(* Logix 5000 project; controller ecust2024 vendor 1 type 14 code 108 rev 30.11; software revision 30.00 *)

TASK MainTask (continuous, watchdog 500 ms) : MainProgram, My_Equipment_Phase

MODULES
   Local : vendor 1 type 14 code 108 (Compact 0, rev 30.11)
      K5500 : 2198-H008-ERS (Ethernet 192.168.1.31, rev 7.13, MotionSync RPI 1 ms, MotionDiagnostics RPI 1 ms)
END_MODULES

ADD_ON_INSTRUCTION AOI   (* revision 1.0 *)
VAR_INPUT
   Start : BOOL; {access None, required}
   Stop : BOOL; {required}
END_VAR
VAR_OUTPUT
   LampOut : BOOL; {access Read Only, required}
END_VAR
VAR_INPUT
   Timer1Set : DINT; {required}
   Timer2Set : DINT; {required}
   Timer3Set : DINT; {required}
   TotalTimerSet : DINT; {required}
END_VAR
VAR
   SysGo : BOOL; {access None}
   Timer_1 : TIMER; {access None}
   Timer_2 : TIMER; {access None}
   Timer_3 : TIMER; {access None}
   Timer_T : TIMER; {access None}
END_VAR

ROUTINE Logic   (* ladder *)
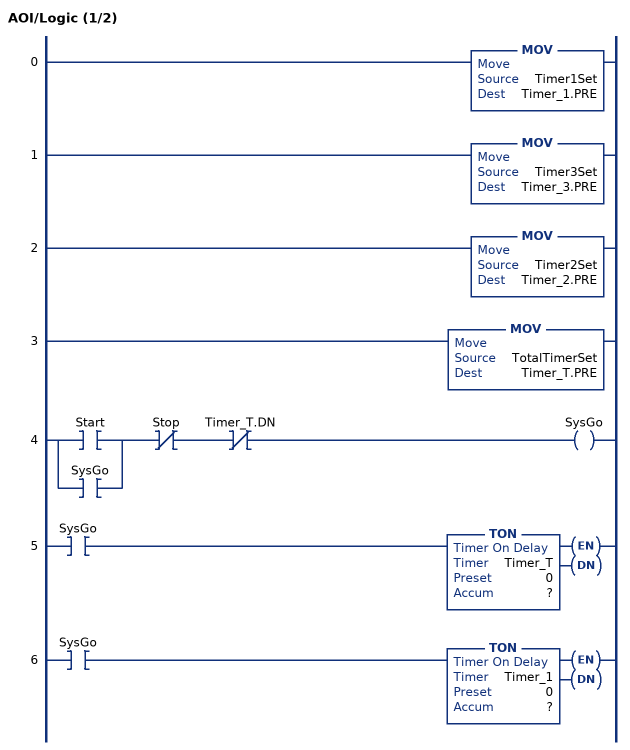
   0: MOV(Timer1Set,Timer_1.PRE);
   1: MOV(Timer3Set,Timer_3.PRE);
   2: MOV(Timer2Set,Timer_2.PRE);
   3: MOV(TotalTimerSet,Timer_T.PRE);
   4: [XIC(Start) ,XIC(SysGo) ]XIO(Stop)XIO(Timer_T.DN)OTE(SysGo);
   5: XIC(SysGo)TON(Timer_T,?,?);
   6: XIC(SysGo)TON(Timer_1,?,?);
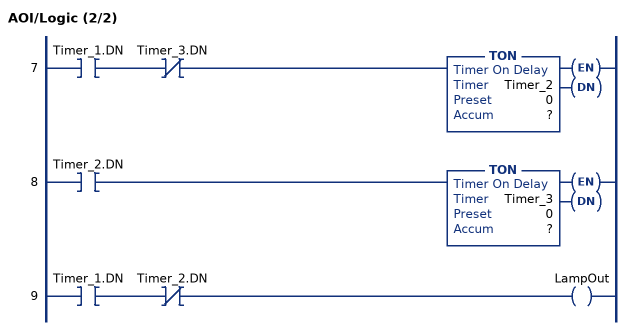
   7: XIC(Timer_1.DN)XIO(Timer_3.DN)TON(Timer_2,?,?);
   8: XIC(Timer_2.DN)TON(Timer_3,?,?);
   9: XIC(Timer_1.DN)XIO(Timer_2.DN)OTE(LampOut);
END_ROUTINE
END_ADD_ON_INSTRUCTION

ADD_ON_INSTRUCTION LED_control   (* revision 1.0 *)
VAR_INPUT
   span : DINT; {required}
END_VAR
VAR_OUTPUT
   LED_start : BOOL; {access Read Only, visible}
END_VAR
VAR_INPUT
   Stop : BOOL; {required}
END_VAR
VAR
   delay1 : TIMER; {access None}
   delay2 : TIMER; {access None}
END_VAR

ROUTINE Logic   (* ladder *)
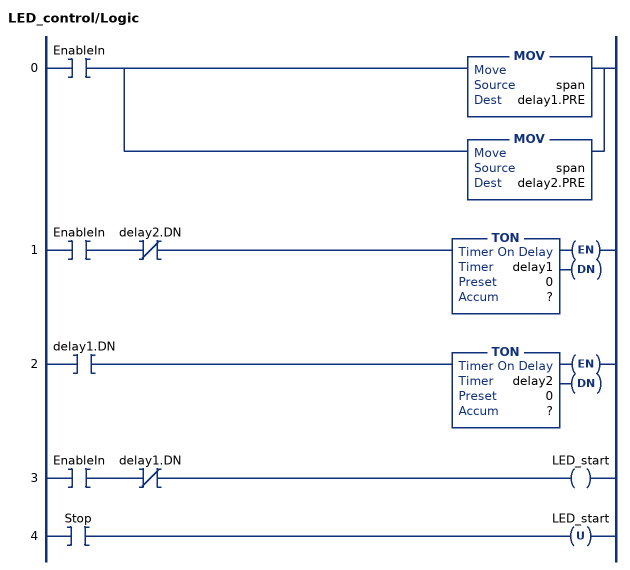
   0: XIC(EnableIn)[MOV(span,delay1.PRE) ,MOV(span,delay2.PRE) ];
   1: XIC(EnableIn)XIO(delay2.DN)TON(delay1,?,?);
   2: XIC(delay1.DN)TON(delay2,?,?);
   3: XIC(EnableIn)XIO(delay1.DN)OTE(LED_start);
   4: XIC(Stop)OTU(LED_start);
END_ROUTINE
END_ADD_ON_INSTRUCTION

ADD_ON_INSTRUCTION OneKey   (* revision 1.0 *)
VAR_INPUT
   Button : BOOL; {required}
END_VAR
VAR_OUTPUT
   On : BOOL; {visible}
   Off : BOOL; {visible}
END_VAR
VAR_INPUT
   Pos1 : DINT; {required}
   Pos2 : DINT; {required}
   speed : DINT; {required}
   Stop_Time : DINT; {required}
END_VAR
VAR_OUTPUT
   Stop1 : BOOL; {access Read Only, visible}
   clockwise : BOOL; {access Read Only, visible}
   anticlockwise : BOOL; {access Read Only, visible}
   Stop2 : BOOL; {access Read Only, visible}
END_VAR
VAR
   delay1 : TIMER; {access None}
   delay2 : TIMER; {access None}
   delay3 : TIMER; {access None}
   oneshot1 : DINT; {access None}
   stop_1 : BOOL; {access None}
   stop_2 : BOOL; {access None}
   Start_state : BOOL; {access None}
   delay4 : TIMER := (PRE := 500); {access None}
END_VAR

ROUTINE Logic   (* ladder *)
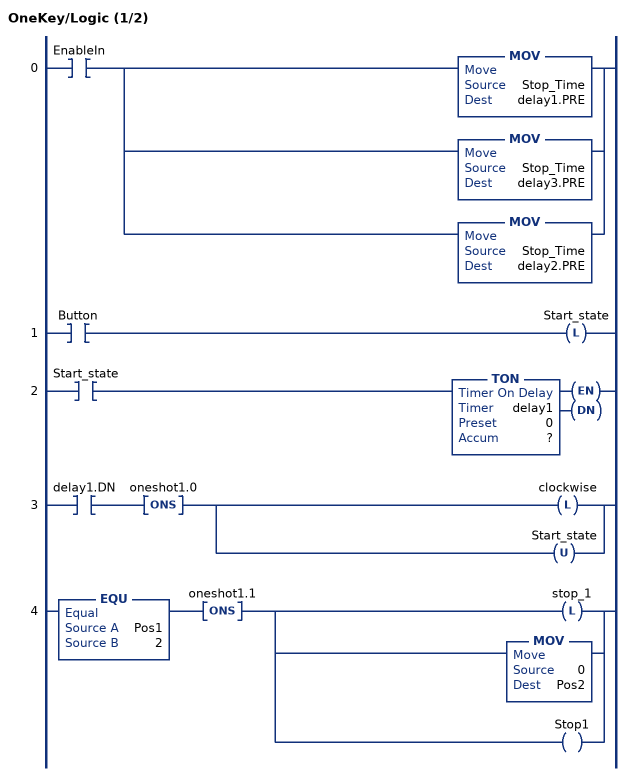
   0: XIC(EnableIn)[MOV(Stop_Time,delay1.PRE) ,MOV(Stop_Time,delay3.PRE) ,MOV(Stop_Time,delay2.PRE) ];
   1: XIC(Button)OTL(Start_state);
   2: XIC(Start_state)TON(delay1,?,?);
   3: XIC(delay1.DN)ONS(oneshot1.0)[OTL(clockwise) ,OTU(Start_state) ];
   4: EQU(Pos1,2)ONS(oneshot1.1)[OTL(stop_1) ,MOV(0,Pos2) ,OTE(Stop1) ];
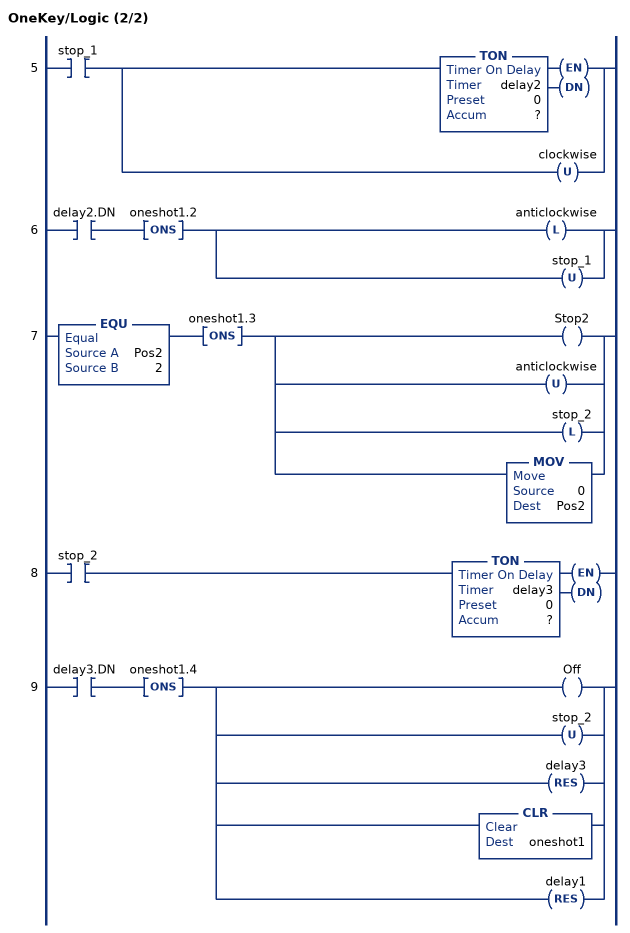
   5: XIC(stop_1)[TON(delay2,?,?) ,OTU(clockwise) ];
   6: XIC(delay2.DN)ONS(oneshot1.2)[OTL(anticlockwise) ,OTU(stop_1) ];
   7: EQU(Pos2,2)ONS(oneshot1.3)[OTE(Stop2) ,OTU(anticlockwise) ,OTL(stop_2) ,MOV(0,Pos2) ];
   8: XIC(stop_2)TON(delay3,?,?);
   9: XIC(delay3.DN)ONS(oneshot1.4)[OTE(Off) ,OTU(stop_2) ,RES(delay3) ,CLR(oneshot1) ,RES(delay1) ];
END_ROUTINE
END_ADD_ON_INSTRUCTION

VAR_GLOBAL   (* controller tags *)
   A : OneKey;
   ActualVelocity_CMX : REAL;
   alrm : BOOL;
   anticlockwise : MOTION_INSTRUCTION := (FLAGS := 570425344, DN := 1);
   anticlockwise2 : MOTION_INSTRUCTION := (FLAGS := 33554432);
   anticlockwise3 : MOTION_INSTRUCTION;
   anticlockwise_order : BOOL;
   Axis_1 : AXIS_CIP_DRIVE;
   back_spot : BOOL;
   backHole : BOOL;
   backHole1_cmd : BOOL;
   backHole1_cmd1 : BOOL := 1;
   backspot : BOOL;
   BletRound : DINT;
   Change_Hole : BOOL;
   Change_speed : BOOL;
   changespeed : MOTION_INSTRUCTION := (FLAGS := 33554432);
   changespeed1 : MOTION_INSTRUCTION := (FLAGS := 33554432);
   changesppedbutton : BOOL;
   circle_num : INT;
   clockwise1 : MOTION_INSTRUCTION := (FLAGS := 570425344, DN := 1);
   clockwise_order : BOOL;
   Cmd_PowerOff : BOOL;
   Cmd_PowerON : BOOL;
   count1 : COUNTER := (PRE := 3);
   count2 : COUNTER := (PRE := 2);
   count3 : COUNTER := (PRE := 2);
   count4 : COUNTER := (PRE := 2);
   count5 : COUNTER := (PRE := 4);
   count6 : COUNTER := (PRE := 4);
   count7 : COUNTER := (PRE := 2);
   count8 : COUNTER := (PRE := 2, ACC := 1);
   countturns1 : TIMER;
   Direction_Change1 : BOOL;
   Direction_Change2 : BOOL;
   Direction_Change3 : BOOL;
   Direction_Change4 : BOOL;
   Direction_change_state1 : BOOL;
   Direction_change_state2 : BOOL;
   Direction_change_state3 : BOOL;
   dong1 : DINT;
   dong2 : DINT;
   Find_sensor1 : BOOL;
   Find_sensor2 : BOOL;
   Find_sensor3 : BOOL;
   Fwd1_Cmd_CMX : BOOL;
   Holding_Cmd : BOOL;
   Light1 : BOOL;
   Light2 : BOOL;
   Light3 : BOOL;
   LT1 : BOOL;
   LT2 : BOOL;
   LT3 : BOOL;
   MSG_1 : MESSAGE;
        MessageParameters(ServiceCode := 16#004c, LocalElement := Temp_CMX, ...)
   MSG_2 : MESSAGE;
        MessageParameters(ServiceCode := 16#004c, LocalElement := Sensor1, ...)
   MSG_3 : MESSAGE;
        MessageParameters(ServiceCode := 16#004c, LocalElement := Sensor2, ...)
   MSG_4 : MESSAGE;
        MessageParameters(ServiceCode := 16#004c, LocalElement := Sensor3, ...)
   My_Equipment_Phase : PHASE := (State := 64, Idle := 1);
   oneshot : DINT;
   Reset_Cmd : BOOL;
   Restart_Cmd : BOOL;
   result1 : DINT;
   result2 : DINT;
   Rev1_Cmd_CMX : BOOL;
   S : DINT;
   screen_speed : DINT := 1;
   Sensor1 : DINT := 1;
   Sensor1_cmd : BOOL := 1;
   Sensor2 : DINT;
   Sensor2_cmd : BOOL;
   Sensor3 : DINT;
   Sensor3_cmd : BOOL;
   Sensor_cmd : BOOL := 1;
   servo_off : MOTION_INSTRUCTION := (FLAGS := 570425344, DN := 1, STATUS := 2, STATE := 1);
   servo_on : MOTION_INSTRUCTION := (FLAGS := 570425344, DN := 1, STATE := 1);
   setspeed : DINT := 1;
   Start_Cmd : BOOL;
   Start_PB : BOOL;
   StartA : BOOL;
   state_fwd : BOOL;
   state_off : BOOL := 1;
   state_on : BOOL;
   state_rev : BOOL;
   state_stop : BOOL;
   Stop : MOTION_INSTRUCTION := (FLAGS := 704643072, DN := 1, PC := 1);
   Stop1 : MOTION_INSTRUCTION := (FLAGS := 33554432);
   Stop1_Cmd_CMX : BOOL;
   Stop2 : MOTION_INSTRUCTION;
   Stop_Cmd : BOOL;
   Stop_PB : BOOL;
   Temp_CMX : REAL;
   temp_speed : REAL;
   temperature_speed : REAL;
   time1 : TIMER := (PRE := 3000);
   time2 : TIMER := (PRE := 3000);
   time3 : TIMER := (PRE := 3000);
   time4 : TIMER := (PRE := 3000);
   ts : BOOL;
   UM_Motion : MOTION_GROUP;
   wendu_alrm : BOOL;
   xiansudu : REAL;
   yanshi1 : TIMER := (PRE := 500);
   yanshi101 : TIMER := (PRE := 3000);
END_VAR

PROGRAM MainProgram   (* main routine MainRoutine *)
VAR
   circle_count : DINT;
   circle_num1 : DINT;
   count10 : COUNTER := (PRE := 3);
   count11 : COUNTER := (PRE := 3);
   delay1 : TIMER := (PRE := 500);
   delay2 : TIMER := (PRE := 1000);
   delay3 : TIMER := (PRE := 1000);
   delay4 : TIMER := (PRE := 1000);
   LED1 : LED_control;
   LED2 : LED_control;
   LED3 : LED_control;
   LT1_AOI : AOI := (Timer2Set := 2000, Timer3Set := 2000, TotalTimerSet := 30000);
   LT2_AOI : AOI := (Timer1Set := 10000, Timer2Set := 1000, Timer3Set := 1000, TotalTimerSet := 30000);
   LT3_AOI : AOI := (Timer1Set := 20000, Timer2Set := 500, Timer3Set := 500, TotalTimerSet := 30000);
   speed_dec : BOOL;
   speed_inc : BOOL;
   velocity : DINT;
   wait1 : TIMER := (PRE := 10000);
   wait2 : TIMER := (PRE := 10000);
   wait3 : TIMER := (PRE := 10000);
END_VAR

ROUTINE MainRoutine   (* ladder *)
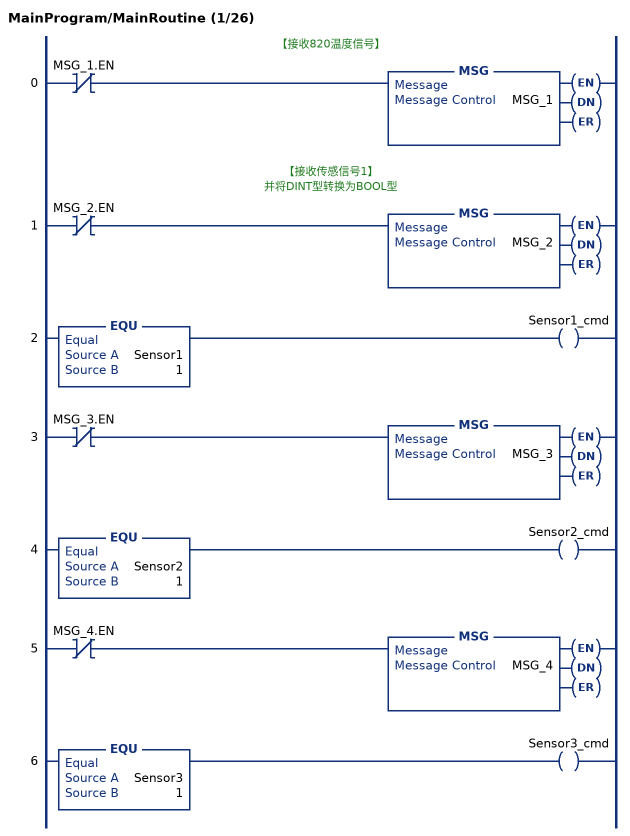
   // 【接收820温度信号】
   0: XIO(MSG_1.EN)MSG(MSG_1);
   // 【接收传感信号1】
   // 并将DINT型转换为BOOL型
   1: XIO(MSG_2.EN)MSG(MSG_2);
   2: EQU(Sensor1,1)OTE(Sensor1_cmd);
   3: XIO(MSG_3.EN)MSG(MSG_3);
   4: EQU(Sensor2,1)OTE(Sensor2_cmd);
   5: XIO(MSG_4.EN)MSG(MSG_4);
   6: EQU(Sensor3,1)OTE(Sensor3_cmd);
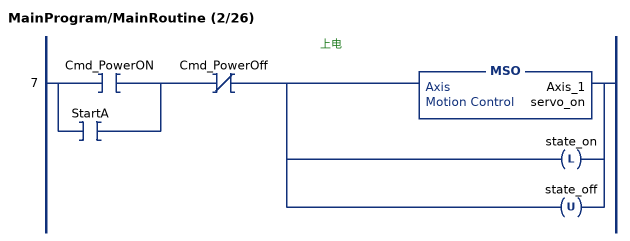
   // 上电
   7: [XIC(Cmd_PowerON) ,XIC(StartA) ]XIO(Cmd_PowerOff)[MSO(Axis_1,servo_on) ,OTL(state_on) ,OTU(state_off) ];
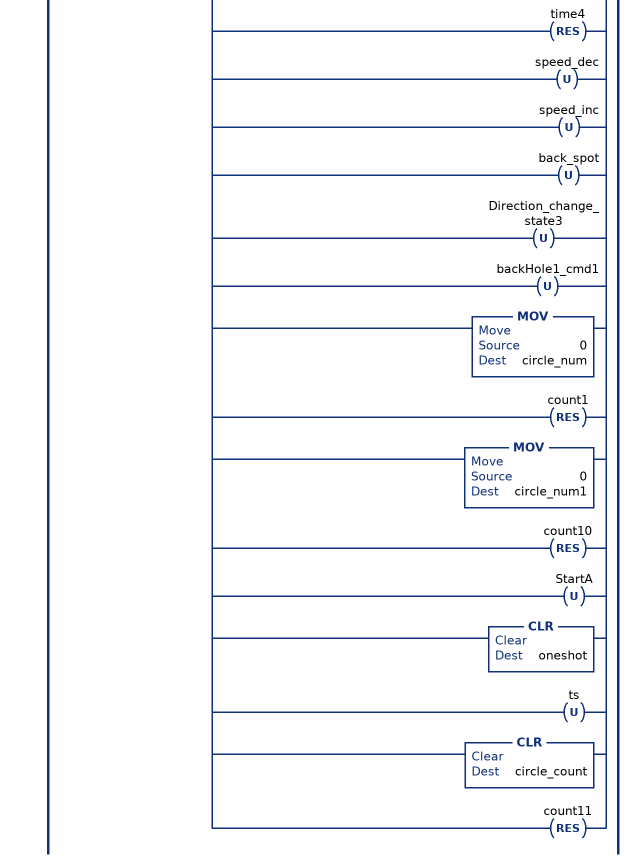
   // 掉电
   // 掉电后，需要置零状态变量
   8: [XIC(Cmd_PowerOff) ,XIC(StartA) XIC(A.Off) ][MSF(Axis_1,servo_off) ,OTU(clockwise_order) ,OTU(anticlockwise_order) ,RES(countturns1) ,OTL(state_off) ,OTU(state_on) ,OTU(state_fwd) ,OTU(state_rev) ,OTU(state_stop) ,OTU(Change_speed) ,MOV(0,ActualVelocity_CMX) ,[MOV(0,BletRound) ,OTU(Direction_change_state1) ,OTU(Direction_Change3) ,OTU(Direction_Change2) ,RES(count5) ,RES(count4) ,RES(count6) ,RES(time4) ,OTU(speed_dec) ,OTU(speed_inc) ,OTU(back_spot) ,OTU(Direction_change_state3) ,OTU(backHole1_cmd1) ,MOV(0,circle_num) ,RES(count1) ,MOV(0,circle_num1) ,RES(count10) ,OTU(StartA) ,CLR(oneshot) ,OTU(ts) ,CLR(circle_count) ,RES(count11) ] ];
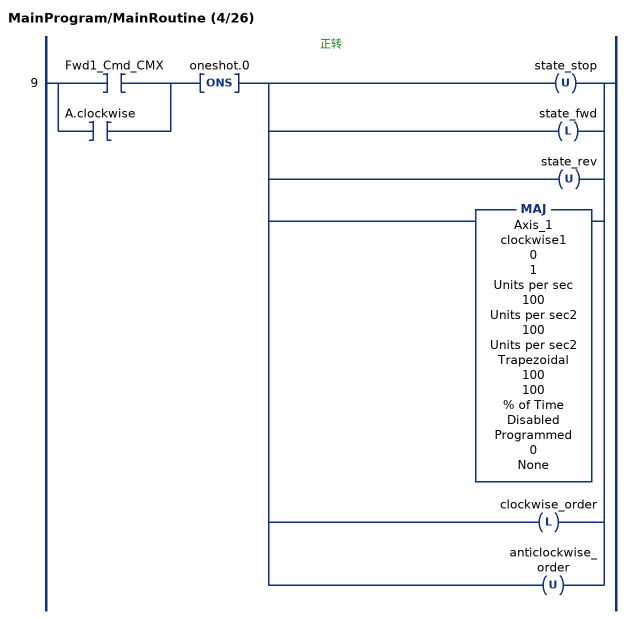
   // 正转
   9: [XIC(Fwd1_Cmd_CMX) ,XIC(A.clockwise) ]ONS(oneshot.0)[OTU(state_stop) ,OTL(state_fwd) ,OTU(state_rev) ,[MAJ(Axis_1,clockwise1,0,1,Units per sec,100,Units per sec2,100,Units per sec2,Trapezoidal,100,100,% of Time,Disabled,Programmed,0,None) ,[OTL(clockwise_order) ,OTU(anticlockwise_order) ] ] ];
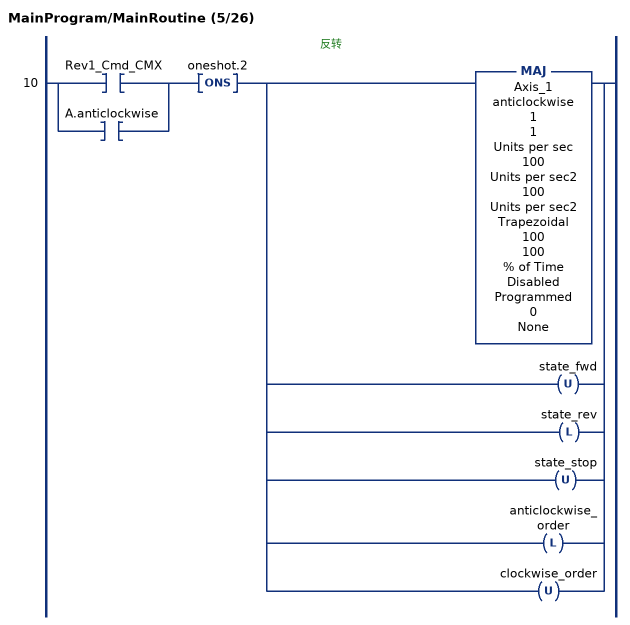
   // 反转
   10: [XIC(Rev1_Cmd_CMX) ,XIC(A.anticlockwise) ]ONS(oneshot.2)[MAJ(Axis_1,anticlockwise,1,1,Units per sec,100,Units per sec2,100,Units per sec2,Trapezoidal,100,100,% of Time,Disabled,Programmed,0,None) ,OTU(state_fwd) ,OTL(state_rev) ,OTU(state_stop) ,OTL(anticlockwise_order) ,OTU(clockwise_order) ];
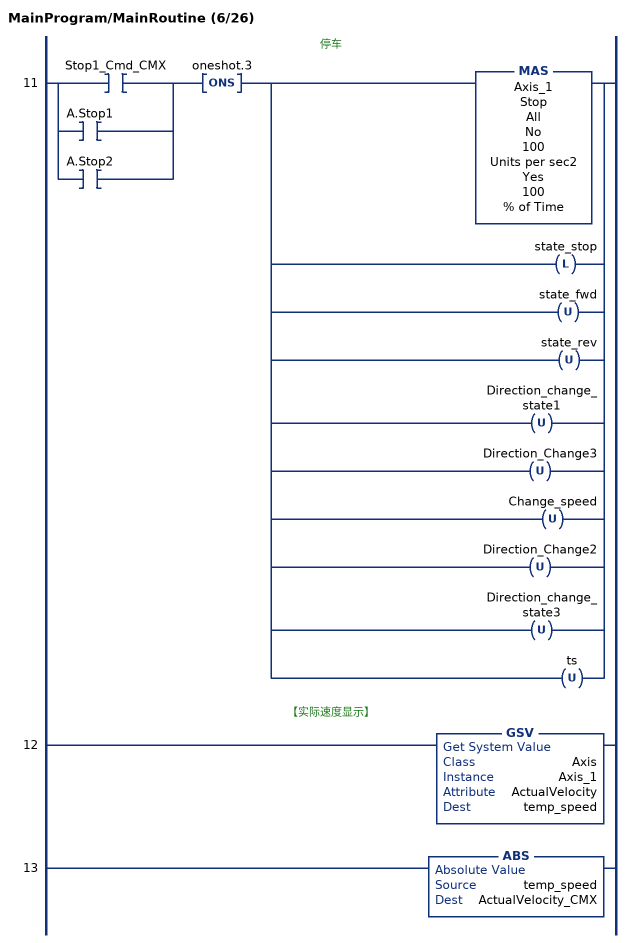
   // 停车
   11: [XIC(Stop1_Cmd_CMX) ,XIC(A.Stop1) ,XIC(A.Stop2) ]ONS(oneshot.3)[MAS(Axis_1,Stop,All,No,100,Units per sec2,Yes,100,% of Time) ,OTL(state_stop) ,OTU(state_fwd) ,OTU(state_rev) ,OTU(Direction_change_state1) ,OTU(Direction_Change3) ,OTU(Change_speed) ,OTU(Direction_Change2) ,OTU(Direction_change_state3) ,OTU(ts) ];
   // 【实际速度显示】
   12: GSV(Axis,Axis_1,ActualVelocity,temp_speed);
   13: ABS(temp_speed,ActualVelocity_CMX);
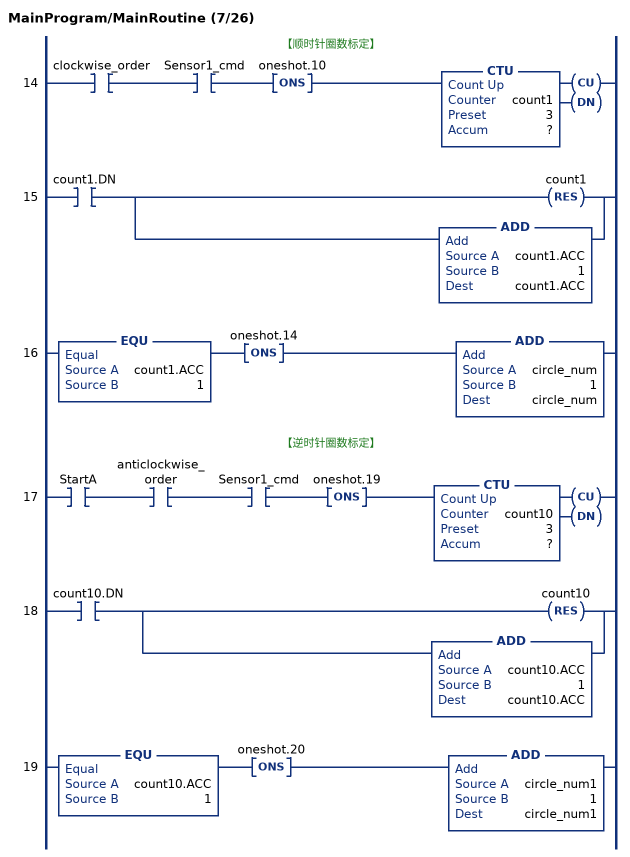
   // 【顺时针圈数标定】
   14: XIC(clockwise_order)XIC(Sensor1_cmd)ONS(oneshot.10)CTU(count1,?,?);
   15: XIC(count1.DN)[RES(count1) ,ADD(count1.ACC,1,count1.ACC) ];
   16: EQU(count1.ACC,1)ONS(oneshot.14)ADD(circle_num,1,circle_num);
   // 【逆时针圈数标定】
   17: XIC(StartA)XIC(anticlockwise_order)XIC(Sensor1_cmd)ONS(oneshot.19)CTU(count10,?,?);
   18: XIC(count10.DN)[RES(count10) ,ADD(count10.ACC,1,count10.ACC) ];
   19: EQU(count10.ACC,1)ONS(oneshot.20)ADD(circle_num1,1,circle_num1);
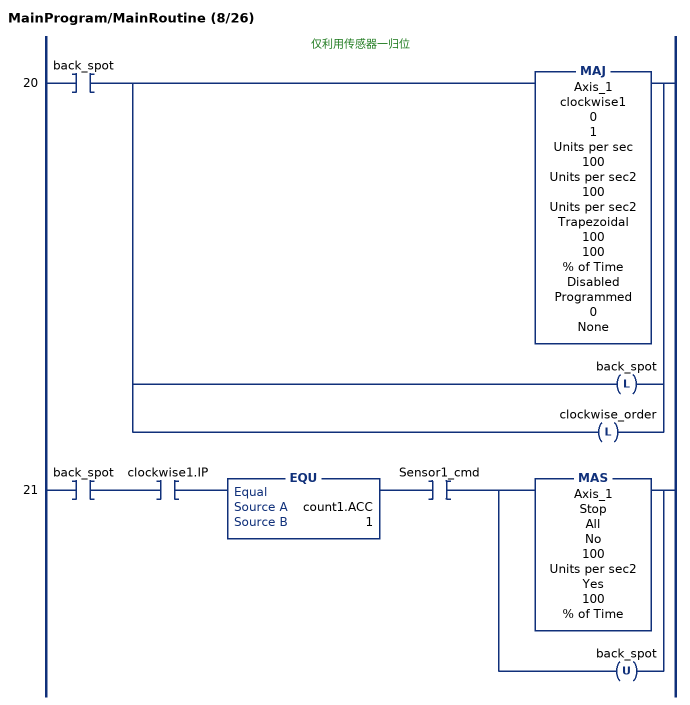
   // 仅利用传感器一归位
   20: XIC(back_spot)[MAJ(Axis_1,clockwise1,0,1,Units per sec,100,Units per sec2,100,Units per sec2,Trapezoidal,100,100,% of Time,Disabled,Programmed,0,None) ,OTL(back_spot) ,OTL(clockwise_order) ];
   21: XIC(back_spot)XIC(clockwise1.IP)EQU(count1.ACC,1)XIC(Sensor1_cmd)[MAS(Axis_1,Stop,All,No,100,Units per sec2,Yes,100,% of Time) ,OTU(back_spot) ];
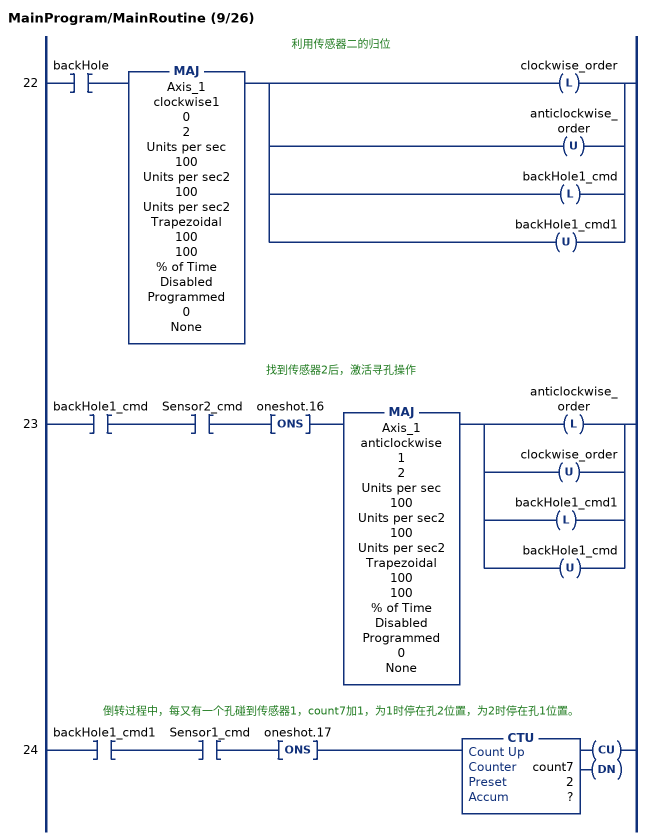
   // 利用传感器二的归位
   22: XIC(backHole)MAJ(Axis_1,clockwise1,0,2,Units per sec,100,Units per sec2,100,Units per sec2,Trapezoidal,100,100,% of Time,Disabled,Programmed,0,None)[OTL(clockwise_order) ,OTU(anticlockwise_order) ,OTL(backHole1_cmd) ,OTU(backHole1_cmd1) ];
   // 找到传感器2后，激活寻孔操作
   23: XIC(backHole1_cmd)XIC(Sensor2_cmd)ONS(oneshot.16)MAJ(Axis_1,anticlockwise,1,2,Units per sec,100,Units per sec2,100,Units per sec2,Trapezoidal,100,100,% of Time,Disabled,Programmed,0,None)[OTL(anticlockwise_order) ,OTU(clockwise_order) ,OTL(backHole1_cmd1) ,OTU(backHole1_cmd) ];
   // 倒转过程中，每又有一个孔碰到传感器1，count7加1，为1时停在孔2位置，为2时停在孔1位置。
   24: XIC(backHole1_cmd1)XIC(Sensor1_cmd)ONS(oneshot.17)CTU(count7,?,?);
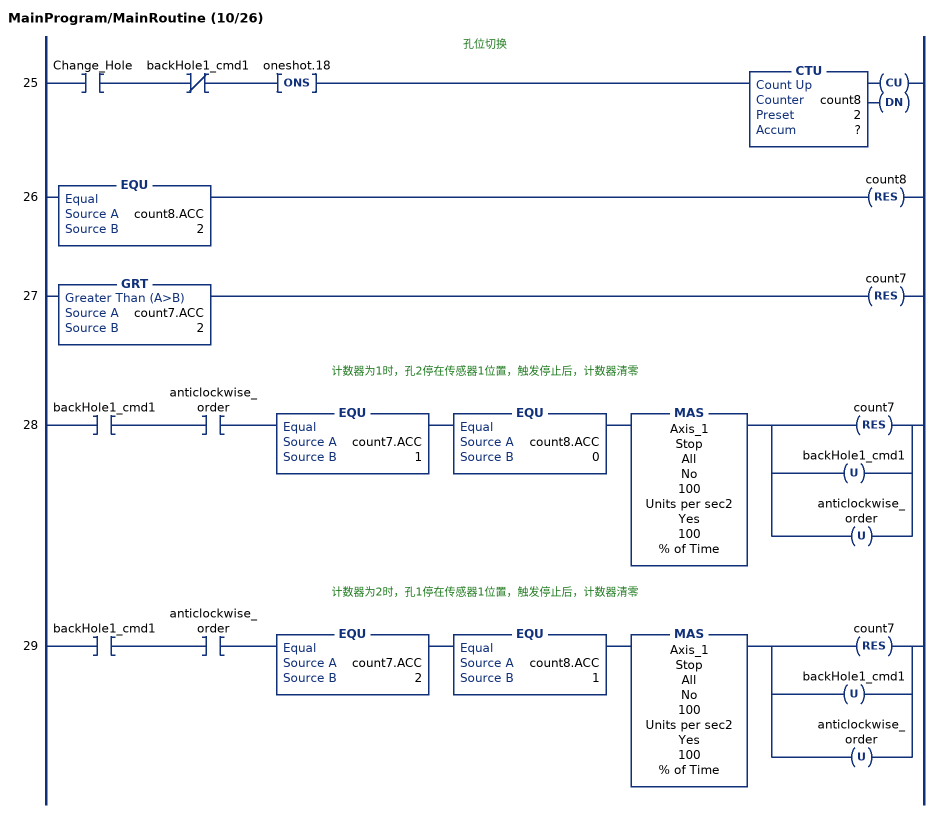
   // 孔位切换
   25: XIC(Change_Hole)XIO(backHole1_cmd1)ONS(oneshot.18)CTU(count8,?,?);
   26: EQU(count8.ACC,2)RES(count8);
   27: GRT(count7.ACC,2)RES(count7);
   // 计数器为1时，孔2停在传感器1位置，触发停止后，计数器清零
   28: XIC(backHole1_cmd1)XIC(anticlockwise_order)EQU(count7.ACC,1)EQU(count8.ACC,0)MAS(Axis_1,Stop,All,No,100,Units per sec2,Yes,100,% of Time)[RES(count7) ,OTU(backHole1_cmd1) ,OTU(anticlockwise_order) ];
   // 计数器为2时，孔1停在传感器1位置，触发停止后，计数器清零
   29: XIC(backHole1_cmd1)XIC(anticlockwise_order)EQU(count7.ACC,2)EQU(count8.ACC,1)MAS(Axis_1,Stop,All,No,100,Units per sec2,Yes,100,% of Time)[RES(count7) ,OTU(backHole1_cmd1) ,OTU(anticlockwise_order) ];
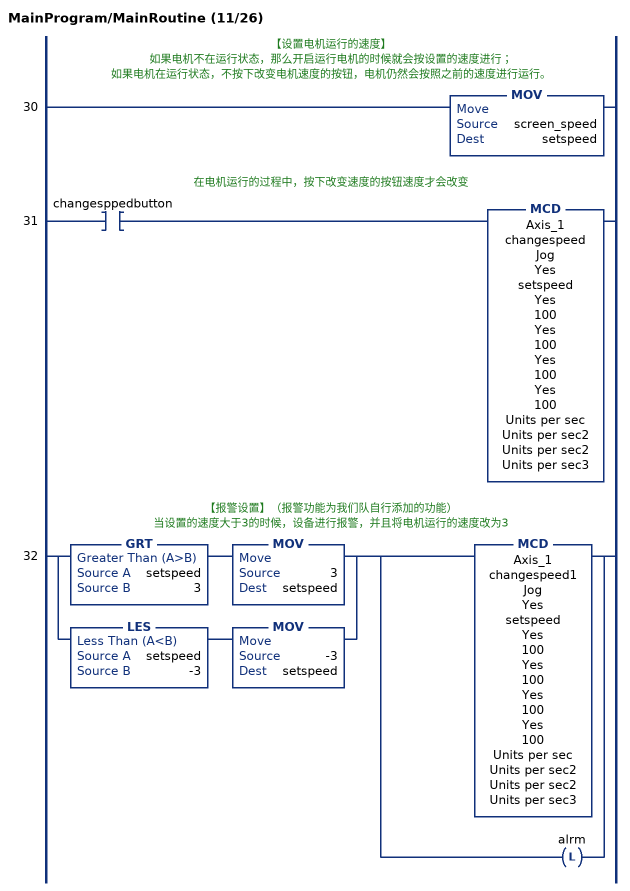
   // 【设置电机运行的速度】
   // 如果电机不在运行状态，那么开启运行电机的时候就会按设置的速度进行；
   // 如果电机在运行状态，不按下改变电机速度的按钮，电机仍然会按照之前的速度进行运行。
   30: MOV(screen_speed,setspeed);
   // 在电机运行的过程中，按下改变速度的按钮速度才会改变
   31: XIC(changesppedbutton)MCD(Axis_1,changespeed,Jog,Yes,setspeed,Yes,100,Yes,100,Yes,100,Yes,100,Units per sec,Units per sec2,Units per sec2,Units per sec3);
   // 【报警设置】（报警功能为我们队自行添加的功能）
   // 当设置的速度大于3的时候，设备进行报警，并且将电机运行的速度改为3
   32: [GRT(setspeed,3) MOV(3,setspeed) ,LES(setspeed,-3) MOV(-3,setspeed) ][MCD(Axis_1,changespeed1,Jog,Yes,setspeed,Yes,100,Yes,100,Yes,100,Yes,100,Units per sec,Units per sec2,Units per sec2,Units per sec3) ,OTL(alrm) ];
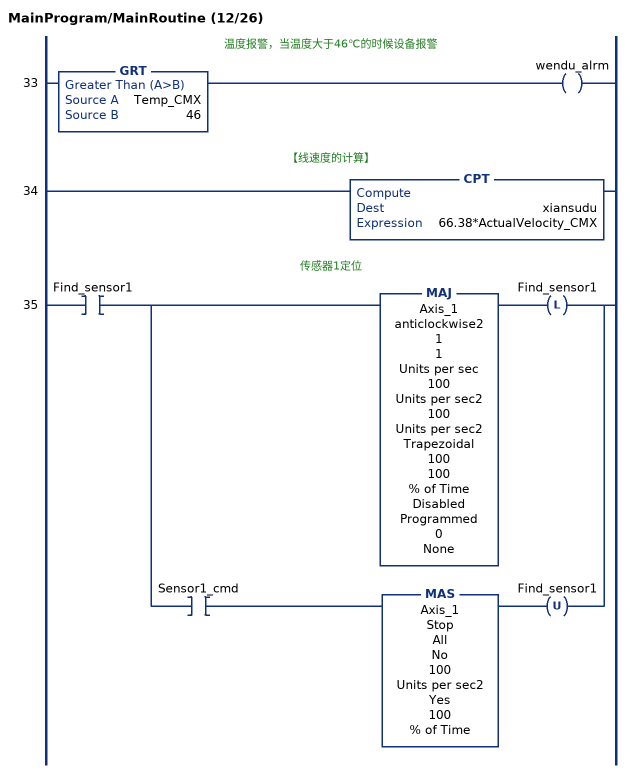
   // 温度报警，当温度大于46℃的时候设备报警
   33: GRT(Temp_CMX,46)OTE(wendu_alrm);
   // 【线速度的计算】
   34: CPT(xiansudu,66.38*ActualVelocity_CMX);
   // 传感器1定位
   35: XIC(Find_sensor1)[MAJ(Axis_1,anticlockwise2,1,1,Units per sec,100,Units per sec2,100,Units per sec2,Trapezoidal,100,100,% of Time,Disabled,Programmed,0,None) OTL(Find_sensor1) ,XIC(Sensor1_cmd) MAS(Axis_1,Stop,All,No,100,Units per sec2,Yes,100,% of Time) OTU(Find_sensor1) ];
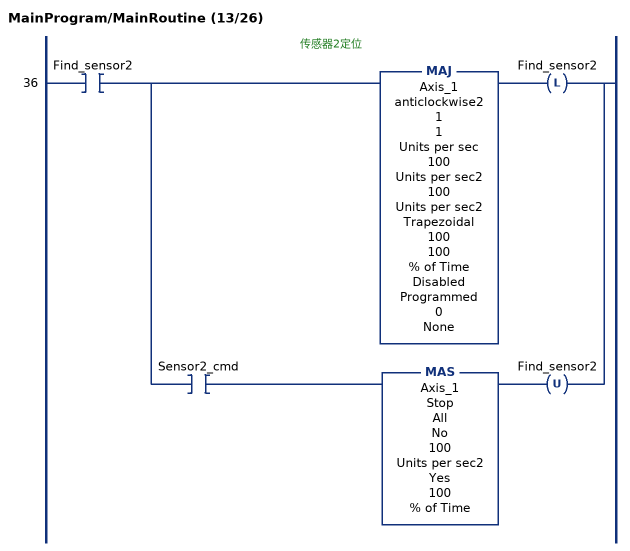
   // 传感器2定位
   36: XIC(Find_sensor2)[MAJ(Axis_1,anticlockwise2,1,1,Units per sec,100,Units per sec2,100,Units per sec2,Trapezoidal,100,100,% of Time,Disabled,Programmed,0,None) OTL(Find_sensor2) ,XIC(Sensor2_cmd) MAS(Axis_1,Stop,All,No,100,Units per sec2,Yes,100,% of Time) OTU(Find_sensor2) ];
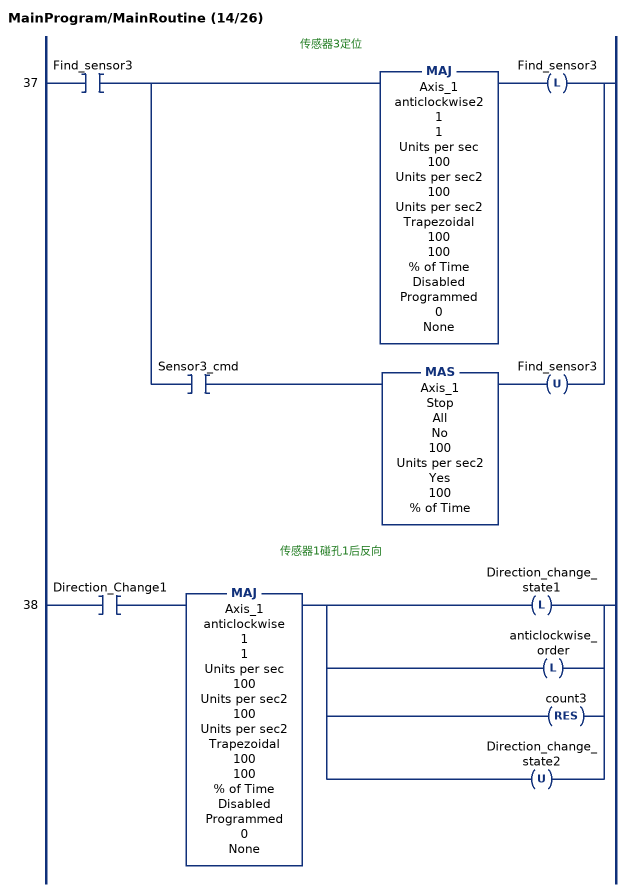
   // 传感器3定位
   37: XIC(Find_sensor3)[MAJ(Axis_1,anticlockwise2,1,1,Units per sec,100,Units per sec2,100,Units per sec2,Trapezoidal,100,100,% of Time,Disabled,Programmed,0,None) OTL(Find_sensor3) ,XIC(Sensor3_cmd) MAS(Axis_1,Stop,All,No,100,Units per sec2,Yes,100,% of Time) OTU(Find_sensor3) ];
   // 传感器1碰孔1后反向
   38: XIC(Direction_Change1)MAJ(Axis_1,anticlockwise,1,1,Units per sec,100,Units per sec2,100,Units per sec2,Trapezoidal,100,100,% of Time,Disabled,Programmed,0,None)[OTL(Direction_change_state1) ,OTL(anticlockwise_order) ,RES(count3) ,OTU(Direction_change_state2) ];
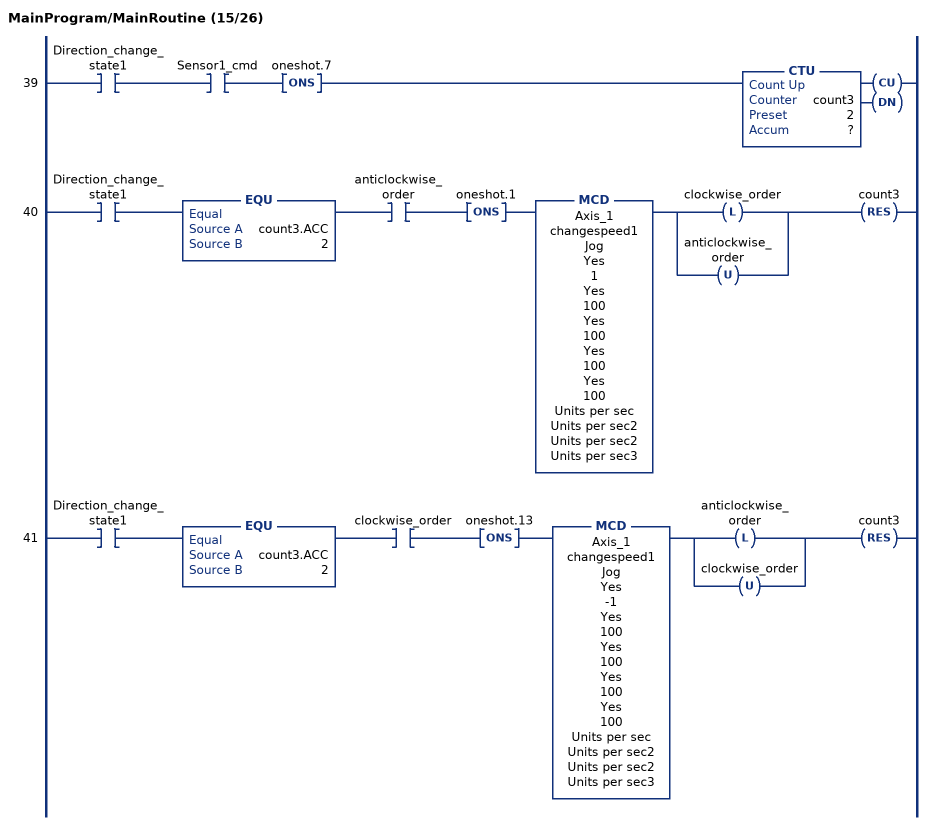
   39: XIC(Direction_change_state1)XIC(Sensor1_cmd)ONS(oneshot.7)CTU(count3,?,?);
   40: XIC(Direction_change_state1)EQU(count3.ACC,2)XIC(anticlockwise_order)ONS(oneshot.1)MCD(Axis_1,changespeed1,Jog,Yes,1,Yes,100,Yes,100,Yes,100,Yes,100,Units per sec,Units per sec2,Units per sec2,Units per sec3)[OTL(clockwise_order) ,OTU(anticlockwise_order) ]RES(count3);
   41: XIC(Direction_change_state1)EQU(count3.ACC,2)XIC(clockwise_order)ONS(oneshot.13)MCD(Axis_1,changespeed1,Jog,Yes,-1,Yes,100,Yes,100,Yes,100,Yes,100,Units per sec,Units per sec2,Units per sec2,Units per sec3)[OTL(anticlockwise_order) ,OTU(clockwise_order) ]RES(count3);
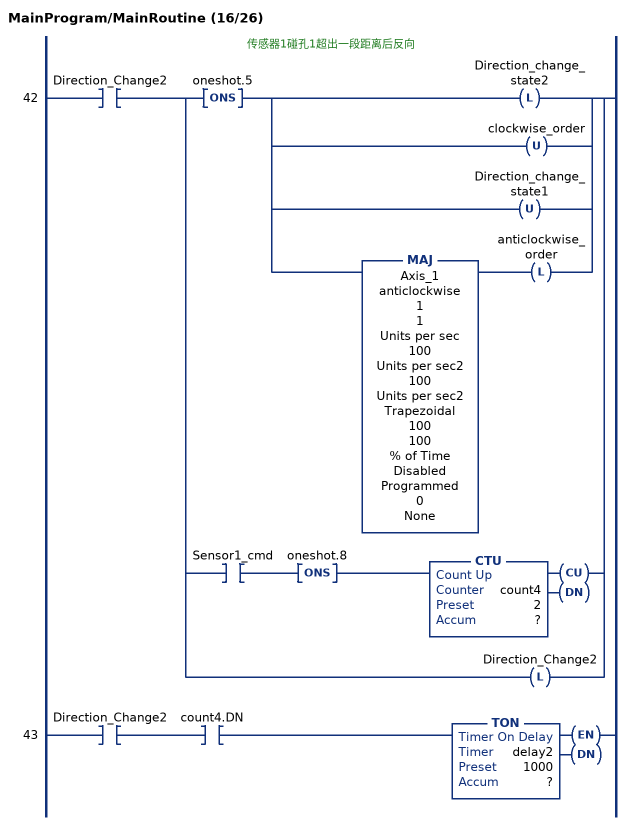
   // 传感器1碰孔1超出一段距离后反向
   42: XIC(Direction_Change2)[ONS(oneshot.5) [OTL(Direction_change_state2) ,OTU(clockwise_order) ,OTU(Direction_change_state1) ,MAJ(Axis_1,anticlockwise,1,1,Units per sec,100,Units per sec2,100,Units per sec2,Trapezoidal,100,100,% of Time,Disabled,Programmed,0,None) OTL(anticlockwise_order) ] ,XIC(Sensor1_cmd) ONS(oneshot.8) CTU(count4,?,?) ,OTL(Direction_Change2) ];
   43: XIC(Direction_Change2)XIC(count4.DN)TON(delay2,?,?);
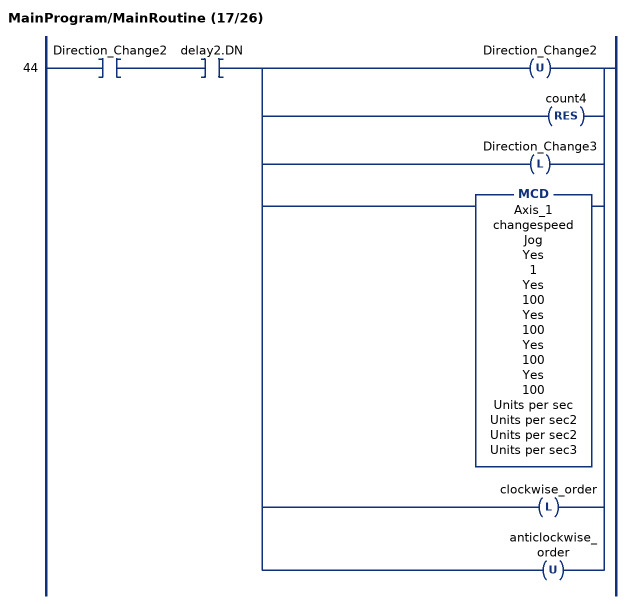
   44: XIC(Direction_Change2)XIC(delay2.DN)[OTU(Direction_Change2) ,RES(count4) ,OTL(Direction_Change3) ,MCD(Axis_1,changespeed,Jog,Yes,1,Yes,100,Yes,100,Yes,100,Yes,100,Units per sec,Units per sec2,Units per sec2,Units per sec3) ,[OTL(clockwise_order) ,OTU(anticlockwise_order) ] ];
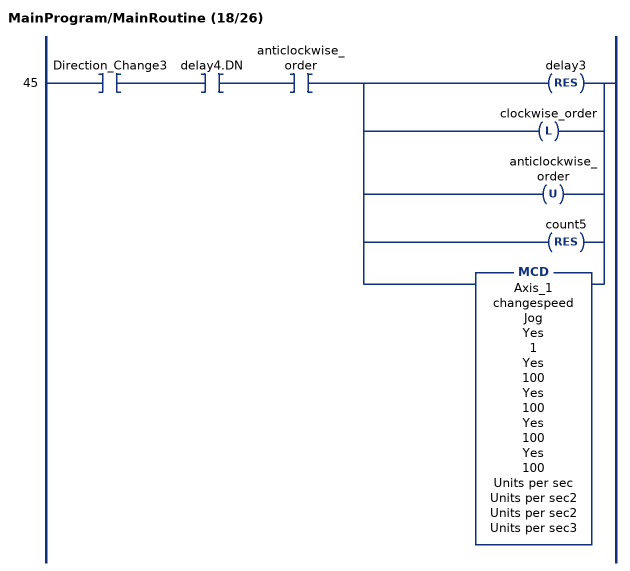
   45: XIC(Direction_Change3)XIC(delay4.DN)XIC(anticlockwise_order)[RES(delay3) ,[OTL(clockwise_order) ,OTU(anticlockwise_order) ,RES(count5) ,MCD(Axis_1,changespeed,Jog,Yes,1,Yes,100,Yes,100,Yes,100,Yes,100,Units per sec,Units per sec2,Units per sec2,Units per sec3) ] ];
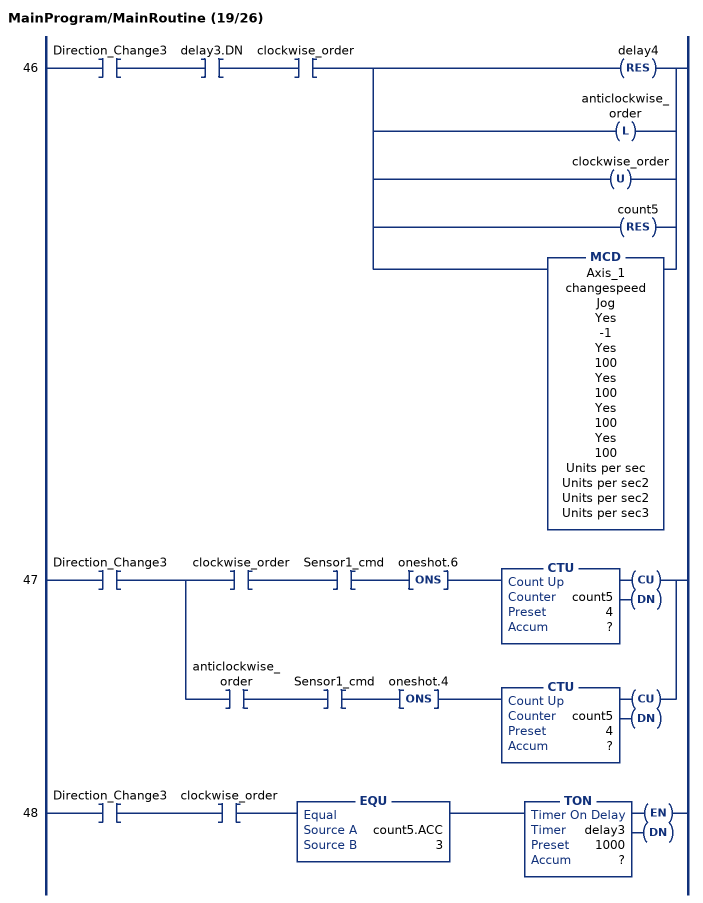
   46: XIC(Direction_Change3)XIC(delay3.DN)XIC(clockwise_order)[RES(delay4) ,OTL(anticlockwise_order) ,OTU(clockwise_order) ,RES(count5) ,MCD(Axis_1,changespeed,Jog,Yes,-1,Yes,100,Yes,100,Yes,100,Yes,100,Units per sec,Units per sec2,Units per sec2,Units per sec3) ];
   47: XIC(Direction_Change3)[XIC(clockwise_order) XIC(Sensor1_cmd) ONS(oneshot.6) CTU(count5,?,?) ,XIC(anticlockwise_order) XIC(Sensor1_cmd) ONS(oneshot.4) CTU(count5,?,?) ];
   48: XIC(Direction_Change3)XIC(clockwise_order)EQU(count5.ACC,3)TON(delay3,?,?);
